Staubli VAL3: start.pgx

program start()
begin
  call MX1_COMMANDS:setup()
  //call MX1_COMMANDS:start()
  call ioLinks()
  taskCreate "network",100,serverCmd()
end
